{attribute 'GeneratedUsingTerminal: EK1122-0000-0018'}
{attribute addProperty BoxType "EK1122-0000-0018"}
{attribute addProperty Id "Beckhoff_EK15xxsub_EK1100EK1100_1FC0878B2A_0001_EK1501_0000_0016EK1501_957D888F6A_0002_EK1501_0000_0017EK1501_957D888F6A_0003_EK1501_0000_0018EK1501_957D888F6A_0004_EK1501_0000_0019EK1501_957D888F6A_0005_EK1501_0010_0016EK1501_957D888F6A_0006_EK1501_0010_0017EK1501_957D888F6A_0007_EK1501_0010_0018EK1501_957D888F6A_0008_EK1501_0100_0016EK1501_957D888F6A_0020_EK1541_0000_0016EK1541_957D888F6A_0021_EK1541_0000_0017EK1541_957D888F6A_0022_EK1541_0000_0018EK1541_957D888F6"}
{attribute addProperty CRC "440552290"}
{attribute addProperty Size "68"}
TYPE Beckhoff_EK15xxEK1122_1A424B62 EXTENDS EK1122_1FC0878B :
STRUCT
	{attribute addProperty Name "Beckhoff_EK15xxsub_EK1100"}
	{attribute addProperty PreviousPort "Beckhoff EK15xxEK1122 : D"}
	Beckhoff_EK15xxsub_EK1100 : EK1100_1FC0878B;
	{attribute addProperty Name "A_0001_EK1501_0000_0016"}
	{attribute addProperty PreviousPort "Beckhoff EK15xxsub EK1100 : C"}
	A_0001_EK1501_0000_0016 : EK1501_957D888F;
	{attribute addProperty Name "A_0002_EK1501_0000_0017"}
	{attribute addProperty PreviousPort "A_0001(EK1501-0000-0016) : C"}
	A_0002_EK1501_0000_0017 : EK1501_957D888F;
	{attribute addProperty Name "A_0003_EK1501_0000_0018"}
	{attribute addProperty PreviousPort "A_0002(EK1501-0000-0017) : C"}
	A_0003_EK1501_0000_0018 : EK1501_957D888F;
	{attribute addProperty Name "A_0004_EK1501_0000_0019"}
	{attribute addProperty PreviousPort "A_0003(EK1501-0000-0018) : C"}
	A_0004_EK1501_0000_0019 : EK1501_957D888F;
	{attribute addProperty Name "A_0005_EK1501_0010_0016"}
	{attribute addProperty PreviousPort "A_0004(EK1501-0000-0019) : C"}
	A_0005_EK1501_0010_0016 : EK1501_957D888F;
	{attribute addProperty Name "A_0006_EK1501_0010_0017"}
	{attribute addProperty PreviousPort "A_0005(EK1501-0010-0016) : C"}
	A_0006_EK1501_0010_0017 : EK1501_957D888F;
	{attribute addProperty Name "A_0007_EK1501_0010_0018"}
	{attribute addProperty PreviousPort "A_0006(EK1501-0010-0017) : C"}
	A_0007_EK1501_0010_0018 : EK1501_957D888F;
	{attribute addProperty Name "A_0008_EK1501_0100_0016"}
	{attribute addProperty PreviousPort "A_0007(EK1501-0010-0018) : C"}
	A_0008_EK1501_0100_0016 : EK1501_957D888F;
	{attribute addProperty Name "A_0020_EK1541_0000_0016"}
	{attribute addProperty PreviousPort "A_0008(EK1501-0100-0016) : C"}
	A_0020_EK1541_0000_0016 : EK1541_957D888F;
	{attribute addProperty Name "A_0021_EK1541_0000_0017"}
	{attribute addProperty PreviousPort "A_0020(EK1541-0000-0016) : C"}
	A_0021_EK1541_0000_0017 : EK1541_957D888F;
	{attribute addProperty Name "A_0022_EK1541_0000_0018"}
	{attribute addProperty PreviousPort "A_0021(EK1541-0000-0017) : C"}
	A_0022_EK1541_0000_0018 : EK1541_957D888F;
END_STRUCT
END_TYPE

(* stored: Version 1.2.0.0, ProductVersion 3.1.4024.9
   DUT Beckhoff_EK15xxEK1122_1A424B62: Id {c38c579e-716f-4427-82a4-5c49a5577b74} *)
